(* IEC 61131-3 sources: com.logicals.lc3.webinar/usRTS_RPMControl_iSOC/src_FB_LIB_SAFE/Safe/Compare, 8 files *)

(* ---- wEQ_SAFEBOOL.iecst ---- *)
NAMESPACE logicals.web.standard.safe
NAMESPACE compare

/*
 * Function block wrapper for IEC 61131-3 EQ<br>
 * IN1 =  1st value (SAFEBOOL)<br>
 * IN2 =  2nd value (SAFEBOOL)<br>
 * OUT = true if IN1 is equal to IN2 (SAFEBOOL)<br>
 */
FUNCTION_BLOCK wEQ_SAFEBOOL
	{ vNameAlignment:="center"; altName:="="; bgColor:="Gold"; width:=40; hideIONames; }
	VAR_INPUT
		IN1 : SAFEBOOL;
		IN2 : SAFEBOOL;
	END_VAR
	VAR_OUTPUT
		OUT : SAFEBOOL;
	END_VAR

	IF (EQ(IN1:=IN1<>SAFEBOOL_Constant#SAFEFALSE, IN2:=IN2<>SAFEBOOL_Constant#SAFEFALSE, ENO=>ENO) <> FALSE)
	THEN
		OUT := SAFEBOOL_Constant#SAFETRUE;
	ELSE
		OUT := SAFEBOOL_Constant#SAFEFALSE;
	END_IF;
	ENO := ENO AND CheckSAFEBOOL(IN1) AND CheckSAFEBOOL(IN2);
END_FUNCTION_BLOCK

END_NAMESPACE
END_NAMESPACE

(* ---- wEQ_SAFEINT.iecst ---- *)
NAMESPACE logicals.web.standard.safe
NAMESPACE compare

/*
 * Function block wrapper for IEC 61131-3 EQ<br>
 * IN1 =  1st value (SAFEINT)<br>
 * IN2 =  2nd value (SAFEINT)<br>
 * OUT = SAFETRUE if IN1 is equal to IN2 (SAFEBOOL)<br>
 */
FUNCTION_BLOCK wEQ_SAFEINT
	{ vNameAlignment:="center"; altName:="="; bgColor:="GoldenRod"; width:=40; hideIONames; }
	VAR_INPUT
		IN1 : SAFEINT;
		IN2 : SAFEINT;
	END_VAR
	VAR_OUTPUT
		OUT : SAFEBOOL;
	END_VAR

	IF (EQ(IN1:=IN1, IN2:=IN2, ENO=>ENO) <> FALSE)
	THEN
		OUT := SAFEBOOL_Constant#SAFETRUE;
	ELSE
		OUT := SAFEBOOL_Constant#SAFEFALSE;
	END_IF;
END_FUNCTION_BLOCK

END_NAMESPACE
END_NAMESPACE

(* ---- wGE_SAFEINT.iecst ---- *)
NAMESPACE logicals.web.standard.safe
NAMESPACE compare

/*
 * Function block wrapper for IEC 61131-3 GE<br>
 * IN1 =  1st value (SAFEINT)<br>
 * IN2 =  2nd value (SAFEINT)<br>
 * OUT = SAFETRUE if IN1 >= IN2 (SAFEBOOL)<br>
 */
FUNCTION_BLOCK wGE_SAFEINT
	{ vNameAlignment:="center"; altName:=">="; bgColor:="GoldenRod"; width:=40; hideIONames; }
	VAR_INPUT
		IN1 : SAFEINT;
		IN2 : SAFEINT;
	END_VAR
	VAR_OUTPUT
		OUT : SAFEBOOL;
	END_VAR

	IF (GE(IN1:=IN1, IN2:=IN2, ENO=>ENO) <> FALSE)
	THEN
		OUT := SAFEBOOL_Constant#SAFETRUE;
	ELSE
		OUT := SAFEBOOL_Constant#SAFEFALSE;
	END_IF;
END_FUNCTION_BLOCK

END_NAMESPACE
END_NAMESPACE

(* ---- wGT_SAFEINT.iecst ---- *)
NAMESPACE logicals.web.standard.safe
NAMESPACE compare

/*
 * Function block wrapper for IEC 61131-3 GT<br>
 * IN1 =  1st value (SAFEINT)<br>
 * IN2 =  2nd value (SAFEINT)<br>
 * OUT = SAFETRUE if IN1 > IN2 (SAFEBOOL)<br>
 */
FUNCTION_BLOCK wGT_SAFEINT
	{ vNameAlignment:="center"; altName:=">"; bgColor:="GoldenRod"; width:=40; hideIONames; }
	VAR_INPUT
		IN1 : SAFEINT;
		IN2 : SAFEINT;
	END_VAR
	VAR_OUTPUT
		OUT : SAFEBOOL;
	END_VAR

	IF (GT(IN1:=IN1, IN2:=IN2, ENO=>ENO) <> FALSE)
	THEN
		OUT := SAFEBOOL_Constant#SAFETRUE;
	ELSE
		OUT := SAFEBOOL_Constant#SAFEFALSE;
	END_IF;
END_FUNCTION_BLOCK

END_NAMESPACE
END_NAMESPACE

(* ---- wLE_SAFEINT.iecst ---- *)
NAMESPACE logicals.web.standard.safe
NAMESPACE compare

/*
 * Function block wrapper for IEC 61131-3 LE<br>
 * IN1 =  1st value (SAFEINT)<br>
 * IN2 =  2nd value (SAFEINT)<br>
 * OUT = SAFETRUE if IN1 <= IN2 (SAFEBOOL)<br>
 */
FUNCTION_BLOCK wLE_SAFEINT
	{ vNameAlignment:="center"; altName:="<="; bgColor:="GoldenRod"; width:=40; hideIONames; }
	VAR_INPUT
		IN1 : SAFEINT;
		IN2 : SAFEINT;
	END_VAR
	VAR_OUTPUT
		OUT : SAFEBOOL;
	END_VAR

	IF (LE(IN1:=IN1, IN2:=IN2, ENO=>ENO) <> FALSE)
	THEN
		OUT := SAFEBOOL_Constant#SAFETRUE;
	ELSE
		OUT := SAFEBOOL_Constant#SAFEFALSE;
	END_IF;
END_FUNCTION_BLOCK

END_NAMESPACE
END_NAMESPACE

(* ---- wLT_SAFEINT.iecst ---- *)
NAMESPACE logicals.web.standard.safe
NAMESPACE compare

/*
 * Function block wrapper for IEC 61131-3 LT<br>
 * IN1 =  1st value (SAFEINT)<br>
 * IN2 =  2nd value (SAFEINT)<br>
 * OUT = SAFETRUE if IN1 < IN2 (SAFEBOOL)<br>
 */
FUNCTION_BLOCK wLT_SAFEINT
	{ vNameAlignment:="center"; altName:="<"; bgColor:="GoldenRod"; width:=40; hideIONames; }
	VAR_INPUT
		IN1 : SAFEINT;
		IN2 : SAFEINT;
	END_VAR
	VAR_OUTPUT
		OUT : SAFEBOOL;
	END_VAR

	IF (LT(IN1:=IN1, IN2:=IN2, ENO=>ENO) <> FALSE)
	THEN
		OUT := SAFEBOOL_Constant#SAFETRUE;
	ELSE
		OUT := SAFEBOOL_Constant#SAFEFALSE;
	END_IF;
END_FUNCTION_BLOCK

END_NAMESPACE
END_NAMESPACE

(* ---- wNE_SAFEBOOL.iecst ---- *)
NAMESPACE logicals.web.standard.safe
NAMESPACE compare

/*
 * Function block wrapper for IEC 61131-3 NE<br>
 * IN1 =  1st value (SAFEBOOL)<br>
 * IN2 =  2nd value (SAFEBOOL)<br>
 * OUT = true if IN1 is not equal to IN2 (SAFEBOOL)<br>
 */
FUNCTION_BLOCK wNE_SAFEBOOL
	{ vNameAlignment:="center"; altName:="<>"; bgColor:="Gold"; width:=40; hideIONames; }
	VAR_INPUT
		IN1 : SAFEBOOL;
		IN2 : SAFEBOOL;
	END_VAR
	VAR_OUTPUT
		OUT : SAFEBOOL;
	END_VAR

	IF (NE(IN1:=IN1<>SAFEBOOL_Constant#SAFEFALSE, IN2:=IN2<>SAFEBOOL_Constant#SAFEFALSE, ENO=>ENO) <> FALSE)
	THEN
		OUT := SAFEBOOL_Constant#SAFETRUE;
	ELSE
		OUT := SAFEBOOL_Constant#SAFEFALSE;
	END_IF;
	ENO := ENO AND CheckSAFEBOOL(IN1) AND CheckSAFEBOOL(IN2);
END_FUNCTION_BLOCK

END_NAMESPACE
END_NAMESPACE

(* ---- wNE_SAFEINT.iecst ---- *)
NAMESPACE logicals.web.standard.safe
NAMESPACE compare

/*
 * Function block wrapper for IEC 61131-3 NE<br>
 * IN1 =  1st value (SAFEINT)<br>
 * IN2 =  2nd value (SAFEINT)<br>
 * OUT = SAFETRUE if IN1 is not equal to IN2 (SAFEBOOL)<br>
 */
FUNCTION_BLOCK wNE_SAFEINT
	{ vNameAlignment:="center"; altName:="<>"; bgColor:="GoldenRod"; width:=40; hideIONames; }
	VAR_INPUT
		IN1 : SAFEINT;
		IN2 : SAFEINT;
	END_VAR
	VAR_OUTPUT
		OUT : SAFEBOOL;
	END_VAR

	IF (NE(IN1:=IN1, IN2:=IN2, ENO=>ENO) <> FALSE)
	THEN
		OUT := SAFEBOOL_Constant#SAFETRUE;
	ELSE
		OUT := SAFEBOOL_Constant#SAFEFALSE;
	END_IF;
END_FUNCTION_BLOCK

END_NAMESPACE
END_NAMESPACE
